TYPE ST_Stepper :
STRUCT
	Axis	:	AXIS_REF;
END_STRUCT
END_TYPE

(* stored: Version 1.1.0.1, ProductVersion 3.1.4020.12
   DUT ST_Stepper: Id {cf35fced-c031-4dfc-8a19-6b35a70ef40a} *)
